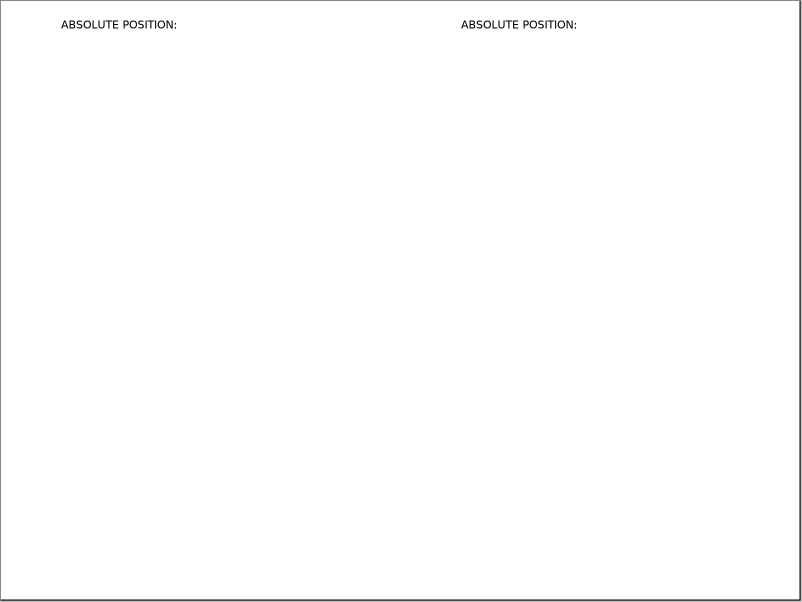
VISUALIZATION F09_Read_Digital_Input  // 802x602
    Rectangle (0,0 800x600)
    Label (10,10 170x30), "ABSOLUTE POSITION:"
    Label (410,10 170x30), "ABSOLUTE POSITION:"
END_VISUALIZATION

(* stored: Version 1.1.0.1, ProductVersion 3.1.4022.7
   Visu F09_Read_Digital_Input: Id {4f71361d-76f7-4303-871d-d2ef265d33bb} *)
